// TIA Portal project "left & right sort" (V16)
// Vorlageprojekt für das Buch mit Zielsystem S7-1200

(* hardware
DEVICE "S7-1200-Station_1"  S7-1200 Station
   slot 0: "Baugruppenträger_0"  Rack  V1.0
   slot 1: "PLC_1"  CPU 1211C DC/DC/DC  6ES7 211-1AE40-0XB0  V4.1
*)

// ===== PLC "PLC_1"  CPU 1211C DC/DC/DC =====

VAR_GLOBAL   // PLC tag table "Standard-Variablentabelle"
   "start" AT %I0.0 : Bool;
   "stop" AT %I0.1 : Bool;
   "turnable1(backlimit)" AT %I0.2 : Bool;
   "turnable1(frontlimit)" AT %I0.3 : Bool;
   "diffuse sensor 1" AT %I1.0 : Bool;
   "diffuse sensor 3" AT %I1.1 : Bool;
   "diffuse sensor 4" AT %I1.2 : Bool;
   "turntable 1 (limit 0)" AT %I1.3 : Bool;
   "turntable 1 (limit 90)" AT %I1.4 : Bool;
   "roller conveyor (4m)1" AT %Q0.0 : Bool;
   "truntable 1 roll (+)" AT %Q0.1 : Bool;
   "truntable 1 turn" AT %Q0.2 : Bool;
   "truntable 1 roll (-)" AT %Q0.3 : Bool;
   "roller conveyor (4m)2" AT %Q0.4 : Bool;
   "roller conveyor (4m)4" AT %Q0.5 : Bool;
   "m1" AT %M0.0 : Bool;
   "m2" AT %M0.1 : Bool;
   "m3" AT %M0.2 : Bool;
   "m4" AT %M0.3 : Bool;
   "m5" AT %M0.4 : Bool;
   "m6" AT %M0.5 : Bool;
   "m7" AT %M0.6 : Bool;
   "m8" AT %M0.7 : Bool;
   "m9" AT %M1.0 : Bool;
   "m10" AT %M1.1 : Bool;
   "m11" AT %M1.2 : Bool;
   "m12" AT %M1.3 : Bool;
   "x1" AT %M1.4 : Bool;
   "x2" AT %M1.5 : Bool;
   "Tag_1" AT %M2.2 : Bool;
   "Tag_2" AT %M3.0 : Bool;
END_VAR

// folder: System blocks/Program resources

DATA_BLOCK "c1"   // DB1
{ S7_Optimized_Access := 'TRUE' }
AUTHOR : Simatic
FAMILY : IEC
NAME : CNTR
VERSION : 1.0
// stored: InstanceOfName IEC_COUNTER
"IEC_COUNTER"
BEGIN
END_DATA_BLOCK

DATA_BLOCK "t1"   // DB2
{ S7_Optimized_Access := 'TRUE' }
AUTHOR : Simatic
FAMILY : IEC
NAME : IEC_TMR
VERSION : 1.0
// stored: InstanceOfName IEC_TIMER
"IEC_TIMER"
BEGIN
END_DATA_BLOCK

// folder: (top level)

FUNCTION "MHJ-PLC-Lab-Function-S71200" : Void   // FC9000, SCL
{ S7_Optimized_Access := 'TRUE' }
VERSION : 0.1
   VAR_TEMP
      rdTimeReturn : Int;
      outputTime : DTL;
      SyncVal : Byte;
      forVal : Int;
      forVal_2 : Int;
      Value : Byte;
   END_VAR
   VAR CONSTANT
      CompVal : Byte := 16#34;
      Value_01 : Byte := 16#11;
      Value_01_DW : DWord := 16#A165_D992;
      Value_02_DW : DWord := 16#58BE_4401;
   END_VAR
BEGIN

   #Value:=PEEK(area := 16#82,
        dbNumber := 0,
        byteOffset := 511);
   #Value := #Value + 1;

   POKE(area := 16#82,
        dbNumber := 0,
        byteOffset := 511,
        value := #Value);

   POKE(area:=16#81,
        dbNumber:=0,
        byteOffset:=1016,
        value:=#Value_01_DW);
   POKE(area := 16#81,
        dbNumber := 0,
        byteOffset := 1020,
        value := #Value_02_DW);

   POKE(area := 16#81,
        dbNumber := 0,
        byteOffset := 511,
        value := B#16#00);

   FOR #forVal := 0 TO 120 DO
       FOR #forVal_2:=0 TO 10 DO
           #rdTimeReturn:=RD_SYS_T(#outputTime);
           #rdTimeReturn := WR_SYS_T(#outputTime);
           #rdTimeReturn := RD_SYS_T(#outputTime);
           #rdTimeReturn := WR_SYS_T(#outputTime);
       END_FOR;
       #SyncVal:= PEEK(area := 16#81,
                      dbNumber := 0,
                      byteOffset := 511);
       IF #SyncVal = #CompVal THEN
          GOTO M_1;
       END_IF;
   END_FOR;
   RETURN;

   M_1:
   POKE(area := 16#81,
        dbNumber := 0,
        byteOffset := 511,
        value := B#16#0);
END_FUNCTION

ORGANIZATION_BLOCK "Main"   // OB1, LAD, ProgramCycle
TITLE = "Main Program Sweep (Cycle)"
{ S7_Optimized_Access := 'TRUE' }
VERSION : 0.1
   VAR_INPUT
      Initial_Call : Bool;   // Initial call of this OB
      Remanence : Bool;   // =True, if remanent data are available
   END_VAR
   VAR_TEMP   // added for the SCL form of the ladder/FBD networks
      _w1 : Bool;
      _w2 : Bool;
   END_VAR
BEGIN

REGION Network 1: Konnektierungsbaustein für PLC-Lab
   // Im Netzwerk 1 wird der Konnektierungsbaustein für PLC-Lab aufgerufen.
   // Dieser Aufruf darf nicht entfernt werden!
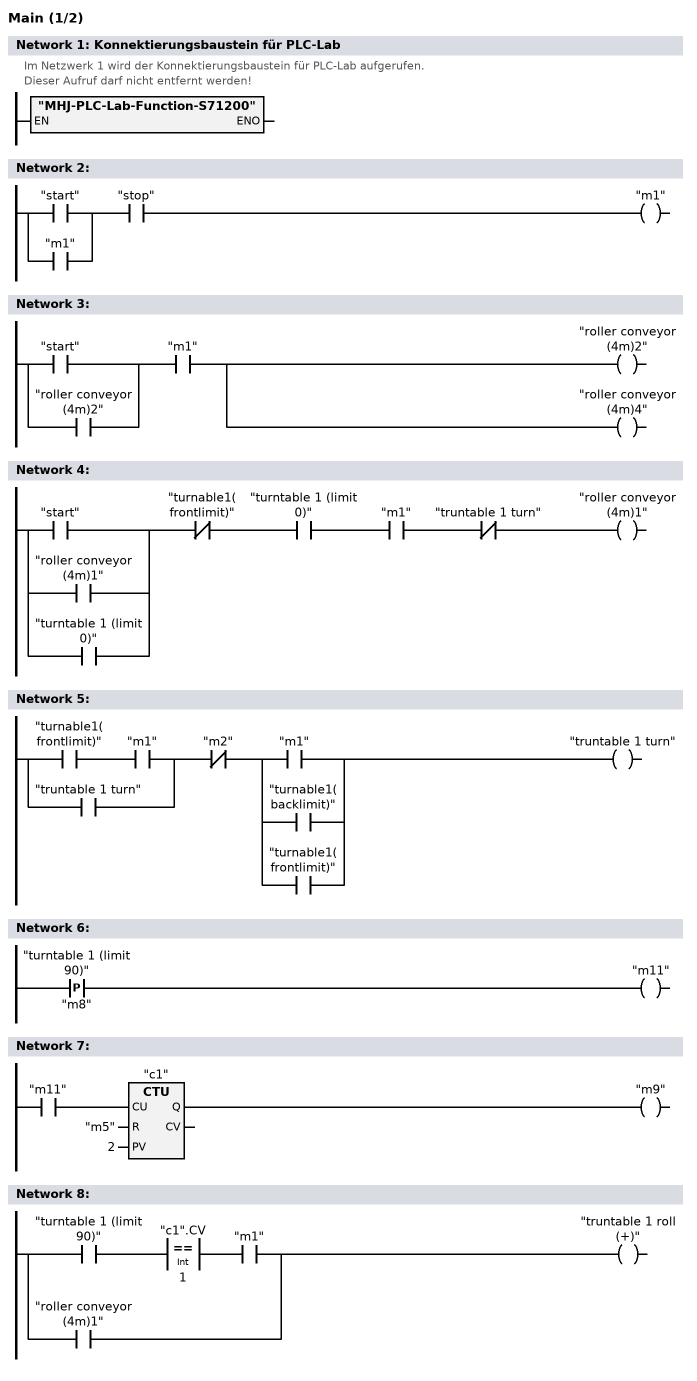
   RUNG wire#powerrail
      "MHJ-PLC-Lab-Function-S71200"()
   END_RUNG
   // the same network as SCL:
   "MHJ-PLC-Lab-Function-S71200"();
END_REGION

REGION Network 2
   RUNG wire#powerrail
      Contact( "start" )
      wire#w1
      Contact( "stop" )
      Coil( "m1" )
   END_RUNG
   RUNG wire#powerrail
      Contact( "m1" )
   END_RUNG wire#w1
   // the same network as SCL:
   "m1" := ("start" OR "m1") AND "stop";
END_REGION

REGION Network 3
   RUNG wire#powerrail
      Contact( "start" )
      wire#w1
      Contact( "m1" )
      wire#w2
      Coil( "roller conveyor (4m)2" )
   END_RUNG
   RUNG wire#powerrail
      Contact( "roller conveyor (4m)2" )
   END_RUNG wire#w1
   RUNG wire#w2
      Coil( "roller conveyor (4m)4" )
   END_RUNG
   // the same network as SCL:
   "roller conveyor (4m)2" := ("start" OR "roller conveyor (4m)2") AND "m1";
   "roller conveyor (4m)4" := "roller conveyor (4m)2";
END_REGION

REGION Network 4
   RUNG wire#powerrail
      Contact( "start" )
      wire#w1
      I_Contact( "turnable1(frontlimit)" )
      Contact( "turntable 1 (limit 0)" )
      Contact( "m1" )
      I_Contact( "truntable 1 turn" )
      Coil( "roller conveyor (4m)1" )
   END_RUNG
   RUNG wire#powerrail
      Contact( "roller conveyor (4m)1" )
   END_RUNG wire#w1
   RUNG wire#powerrail
      Contact( "turntable 1 (limit 0)" )
   END_RUNG wire#w1
   // the same network as SCL:
   "roller conveyor (4m)1" := ("start" OR "roller conveyor (4m)1" OR "turntable 1 (limit 0)") AND NOT "turnable1(frontlimit)" AND "turntable 1 (limit 0)" AND "m1" AND NOT "truntable 1 turn";
END_REGION

REGION Network 5
   RUNG wire#powerrail
      Contact( "turnable1(frontlimit)" )
      Contact( "m1" )
      wire#w1
      I_Contact( "m2" )
      wire#w2
      Contact( "m1" )
      wire#w3
      Coil( "truntable 1 turn" )
   END_RUNG
   RUNG wire#powerrail
      Contact( "truntable 1 turn" )
   END_RUNG wire#w1
   RUNG wire#w2
      Contact( "turnable1(backlimit)" )
   END_RUNG wire#w3
   RUNG wire#w2
      Contact( "turnable1(frontlimit)" )
   END_RUNG wire#w3
   // the same network as SCL:
   "truntable 1 turn" := (("turnable1(frontlimit)" AND "m1") OR "truntable 1 turn") AND NOT "m2" AND ("m1" OR "turnable1(backlimit)" OR "turnable1(frontlimit)");
END_REGION

REGION Network 6
   RUNG wire#powerrail
      P_Contact(operand := "turntable 1 (limit 90)", bit := "m8")
      Coil( "m11" )
   END_RUNG
   // the same network as SCL:
   #_w1 := "turntable 1 (limit 90)" AND NOT "m8";   // rising edge of "turntable 1 (limit 90)"
   "m8" := "turntable 1 (limit 90)";
   "m11" := #_w1;
END_REGION

REGION Network 7
   "c1".CTU(CU := "m11", R := "m5", PV := 2);
   "m9" := "c1".Q;
END_REGION

REGION Network 8
   RUNG wire#powerrail
      Contact( "turntable 1 (limit 90)" )
      { S7_Templates := "SrcType := Int" } EQ_Contact(in1 := "c1".CV, in2 := 1)
      Contact( "m1" )
      wire#w1
      Coil( "truntable 1 roll (+)" )
   END_RUNG
   RUNG wire#powerrail
      Contact( "roller conveyor (4m)1" )
   END_RUNG wire#w1
   // the same network as SCL:
   "truntable 1 roll (+)" := ("turntable 1 (limit 90)" AND ("c1".CV = 1) AND "m1") OR "roller conveyor (4m)1";
END_REGION

REGION Network 9
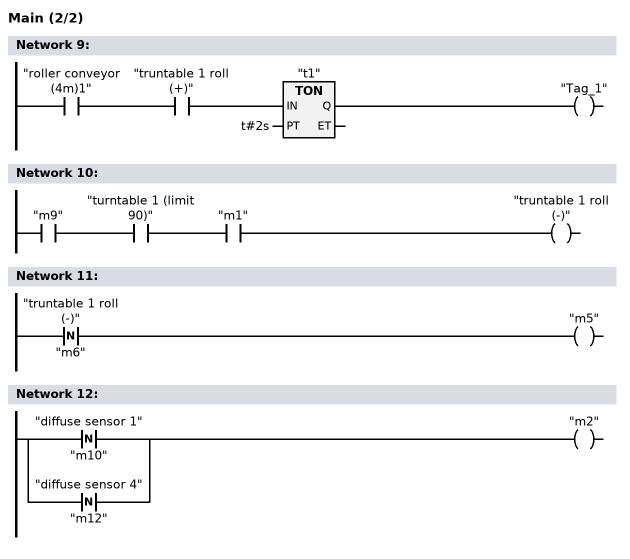
   "t1".TON(IN := "roller conveyor (4m)1" AND "truntable 1 roll (+)", PT := t#2s);
   "Tag_1" := "t1".Q;
END_REGION

REGION Network 10
   RUNG wire#powerrail
      Contact( "m9" )
      Contact( "turntable 1 (limit 90)" )
      Contact( "m1" )
      Coil( "truntable 1 roll (-)" )
   END_RUNG
   // the same network as SCL:
   "truntable 1 roll (-)" := "m9" AND "turntable 1 (limit 90)" AND "m1";
END_REGION

REGION Network 11
   RUNG wire#powerrail
      N_Contact(operand := "truntable 1 roll (-)", bit := "m6")
      Coil( "m5" )
   END_RUNG
   // the same network as SCL:
   #_w1 := NOT "truntable 1 roll (-)" AND "m6";   // falling edge of "truntable 1 roll (-)"
   "m6" := "truntable 1 roll (-)";
   "m5" := #_w1;
END_REGION

REGION Network 12
   RUNG wire#powerrail
      N_Contact(operand := "diffuse sensor 1", bit := "m10")
      wire#w1
      Coil( "m2" )
   END_RUNG
   RUNG wire#powerrail
      N_Contact(operand := "diffuse sensor 4", bit := "m12")
   END_RUNG wire#w1
   // the same network as SCL:
   #_w1 := NOT "diffuse sensor 1" AND "m10";   // falling edge of "diffuse sensor 1"
   "m10" := "diffuse sensor 1";
   #_w2 := NOT "diffuse sensor 4" AND "m12";   // falling edge of "diffuse sensor 4"
   "m12" := "diffuse sensor 4";
   "m2" := #_w1 OR #_w2;
END_REGION
END_ORGANIZATION_BLOCK